FUNCTION_BLOCK FB_Moving_average
VAR_INPUT
	New_sample: REAL;
	Num_samples: INT;
END_VAR
VAR_OUTPUT
	Out: REAL;
END_VAR
VAR CONSTANT
	Array_size: INT := 300;	
END_VAR
VAR
	Samples: ARRAY[0..(Array_size - 1)] OF REAL;
	i: INT;
	Sum: REAL;
END_VAR

Sum:= 0;
FOR i :=

END_FUNCTION_BLOCK

(* stored: Version 1.1.0.1, ProductVersion 3.1.4024.0
   POU FB_Moving_average: Id {2e1d2178-5453-438c-919f-53b5a6335811}, SpecialFunc None *)
